Fanuc KAREL source: ka00132.KL

-- PROVISIONAL review KL for V940-1; original PC SHA256 7b70311836103261817d06fb437507621ff77c5ff45578aec254fe96a2e62820
-- Incomplete behavior may be omitted. Consult companion uncertainty JSON. Do not deploy.
PROGRAM KA00132
%NOLOCKGROUP
-- UNRESOLVED_DECL SRC type=002018
-- UNRESOLVED_DECL DST type=002017
BEGIN
  -- V9_ZERO_TABLE_METADATA_HINT layout=0001; no indexed target words; source/name/runtime held
  -- UNRESOLVED_PC offsets 5-19; opcodes 2E,22,9D,33,B2
  -- UNRESOLVED_PC offsets 24-42; opcodes 22,9D,33,B1,22,9D,33,B4
  -- UNRESOLVED_PC offsets 47-51; opcodes 7F
END KA00132
